FUNCTION_BLOCK Power_lever
VAR_INPUT
END_VAR
VAR_OUTPUT
END_VAR
VAR
END_VAR

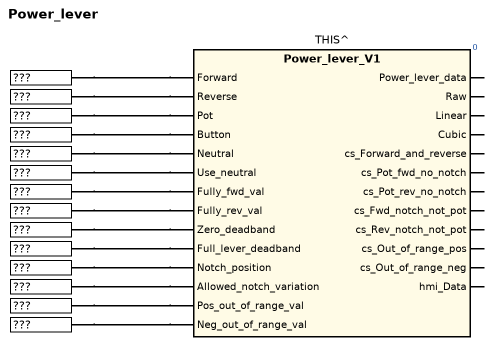
THIS^(
    Forward := ???,
    Reverse := ???,
    Pot := ???,
    Button := ???,
    Neutral := ???,
    Use_neutral := ???,
    Fully_fwd_val := ???,
    Fully_rev_val := ???,
    Zero_deadband := ???,
    Full_lever_deadband := ???,
    Notch_position := ???,
    Allowed_notch_variation := ???,
    Pos_out_of_range_val := ???,
    Neg_out_of_range_val := ???); // Power_lever_V1

METHOD Power_lever_V1
VAR_INPUT
	Forward:BOOL; (*Lever notch 1 forward*)
	Reverse:BOOL; (*Lever notch 1 reverse*)
	Pot:INT; (*Analogue value from lever potentiometer*)
	Button:BOOL;
	
	Neutral:BOOL;
	Use_neutral:BOOL;
	
	Fully_fwd_val:INT; (*Value of analogue input when lever is fully forward*)
	Fully_rev_val:INT; (*Value of analogue input when lever is fully reverse*)
	Zero_deadband:INT; (*Lever zero position deadband on a scale of 0 to 10 000 i.e. a value of 100 gives a 1% deadband in each direction*)
	Full_lever_deadband:INT; (*Lever fully forward or reverse deadband on a scale of 0 to 10 000 i.e. a value of 100 gives a 1% deadband*)
	
	Notch_position:INT; (*Lever value (-10 000 to 10 000, no deadbands) at which forward and reverse notches change state*)
	Allowed_notch_variation:INT; (*Allowed variation in notch position*)
	Pos_out_of_range_val:INT; (*If the analogue Pot value exceeds this threshold, a fault will be generated.*)
	Neg_out_of_range_val:INT; (*If the analogue Pot value is less than this threshold, a fault will be generated.*)
END_VAR
VAR_OUTPUT
	Power_lever_data:dut_Power_lever; (*Power lever data packed into a single structure.*)
	
	Raw:INT; (*Linear scaled lever value with no deadbands applied. -10 000 = fully reverse. +10 000 = fully forward.*)
	Linear:INT;
	Cubic:INT;
	
	cs_Forward_and_reverse:BOOL;
	cs_Pot_fwd_no_notch:BOOL;
	cs_Pot_rev_no_notch:BOOL;
	cs_Fwd_notch_not_pot:BOOL;
	cs_Rev_notch_not_pot:BOOL;
	cs_Out_of_range_pos:BOOL;
	cs_Out_of_range_neg:BOOL;
	
	hmi_Data:dut_hmi_Power_lever;
END_VAR
END_METHOD

END_FUNCTION_BLOCK

(* stored: Version 1.1.0.1, ProductVersion 3.1.4024.0
   POU Power_lever: Id {0c6f5f18-597a-4fda-9fcd-6cc2ed86d36c}, SpecialFunc None
   Method Power_lever_V1: Id {562e64b3-7dc0-4477-b51a-082414aec197} *)
